// TIA Portal V16 export
// export: Created 2024-12-03T15:41:45.7500628Z, ExportSetting WithReadOnly, DisplayName Totally Integrated Automation Portal, DisplayVersion V16 Update 6, DisplayName TIA Portal Version Control Interface, DisplayVersion V16 Update 2, DisplayName TIA Portal Openness, DisplayVersion V16 Update 6, DisplayName TIA Portal Teamcenter Gateway, DisplayVersion V16, DisplayName SINAMICS Startdrive Advanced, DisplayVersion V16 Update 5, DisplayName SINAMICS Startdrive G130, G150, S120, S150, SINAMICS MV, S210, DisplayVersion V16 Update 5, DisplayName SINAMICS Startdrive G110M, G120, G120C, G120D, G120P, G115D, DisplayVersion V16 Update 5, DisplayName STEP 7 Professional, DisplayVersion V16 Update 6, DisplayName STEP 7 Safety, DisplayVersion V16, DisplayName WinCC Advanced / Unified PC, DisplayVersion V16 Update 6
TYPE "SKTU4_In_Data_UDT"
// stored: CreationDate 2023-04-19T11:30:38.0051651Z, InterfaceModifiedDate 2023-04-19T12:03:36.2470411Z, IsConsistent true, LibraryConformanceStatus The object is library-conformant., ModifiedDate 2023-04-19T12:03:36.2470411Z
   STRUCT
      reserve7 : Byte;
      Input_1 : Bool;
      Input_2 : Bool;
      Input_3 : Bool;
      Input_4 : Bool;
      Input_5 : Bool;
      Input_6 : Bool;
      Input_7 : Bool;
      Input_8 : Bool;
   END_STRUCT;
END_TYPE
